ABB RobotStudio station: PickAndPlace_ManipulatorRobot.rspag

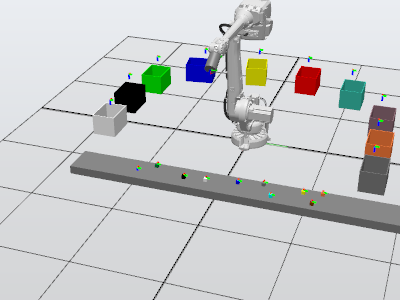
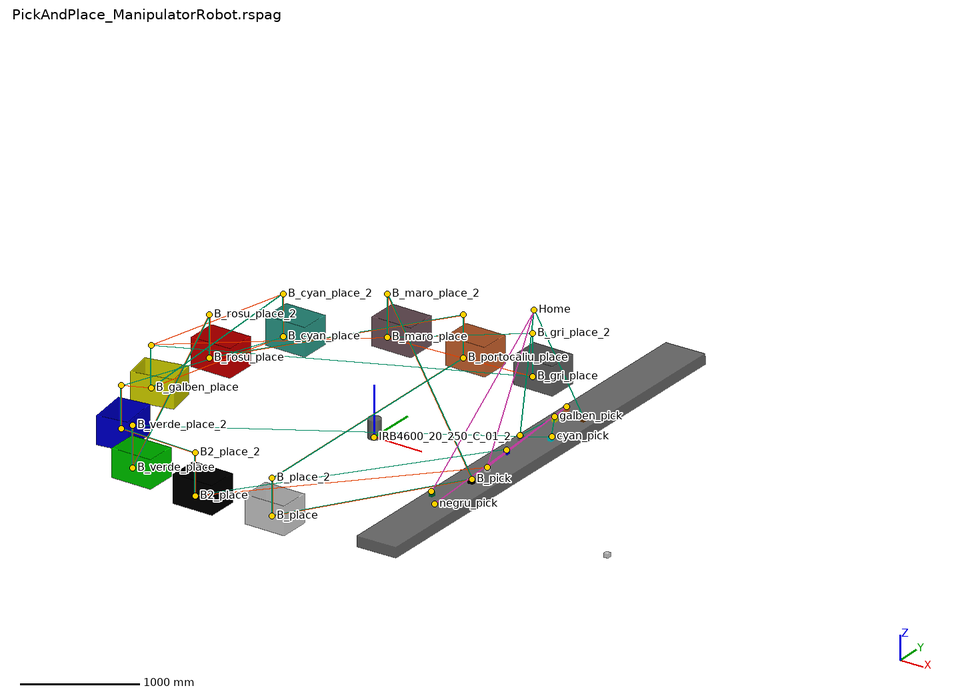
[picture v1: parts stored in the station drawn from their meshes, with robot base, taught points and paths (robot models come from the ABB library and are not in the file)]
--- station ---
Station Tema1 (saved by RobotStudio 24.3.10958.1)
Controller Controller1
  mechanical unit ROB_1: IRB4600_20_250_C_01_2, 6 joints, base frame (0, 0, 0) mm
Layout (positions relative to the parent item):
  - Container [part] at (-1892.47, -1896.95, 0) mm, size 400 x 300 x 270 mm
  - Container_2 [part] at (-161.95, 1479.58, 0) mm, size 400 x 300 x 270 mm
  - Container_4 [part] at (-1211.54, -114.6, 0) mm, rotated rx 0 ry 0 rz -168.57 deg, size 400 x 300 x 270 mm
  - Container_5 [part] at (-1951.65, -525.59, 0) mm, rotated rx 0 ry 0 rz -82.41 deg, size 400 x 300 x 270 mm
  - Cutia_alba [part] at (-473.04, -1981.87, 0) mm, size 400 x 300 x 270 mm
  - Container_7 [part] at (-1188.6, -2007.67, 0) mm, size 400 x 300 x 270 mm
  - Container_8 [part] at (-1549.29, 1401.48, 0) mm, size 400 x 300 x 270 mm
  - Container_9 [part] at (-2281.34, 903.83, 0) mm, size 400 x 300 x 270 mm
  - Container_10 [part] at (-2561.63, 214.84, 0) mm, size 400 x 300 x 270 mm
  - Banda Transport [part] at (1467.9, -1784.42, 101.57) mm, rotated rx -180 ry 0.95 rz -180 deg, size 400 x 4500 x 100 mm
  - Container_11 [part] at (-833.57, 1452.99, 0) mm, size 400 x 300 x 270 mm
  - griper [mechanism] at (1479.11, 0, 1722.5) mm, rotated rx -180 ry 60 rz -180 deg
      TCP griper at (0, 0, 175) mm
      links: Part_3
  - orn [part] at (2566.83, 0, 745.86) mm, size 40 x 40 x 40 mm
  - cutia_neagra-alb [part] at (1281.21, -423.55, 138.52) mm, rotated rx 180 ry 0 rz 180 deg, size 40 x 40 x 40 mm
  - alba [part] at (1269.69, -164.67, 139.56) mm, rotated rx 180 ry 0 rz 180 deg, size 40 x 40 x 40 mm
  - albastra [part] at (1207.67, 200.37, 140.96) mm, rotated rx 180 ry 0 rz 180 deg, size 40 x 40 x 40 mm
  - cyan [part] at (1364.48, 621.04, 140.84) mm, rotated rx 180 ry 0 rz 180 deg, size 40 x 40 x 40 mm
  - galben [part] at (1176.16, 945.56, 137.64) mm, rotated rx 180 ry 0 rz 180 deg, size 40 x 40 x 40 mm
  - rosu [part], size 40 x 40 x 40 mm
  - IRB4600_20_250_C_01_2 [mechanism, from %ABB.RobotStudio.Models.IRB4600%\IRB4600_20_250_C_G_01.rslib] at (0, 0, 0) mm; joint values [0, 0, 0, 0, 0.5236, 0] (rad or m)
  - ComponentInstance [part], size 120 x 119.8 x 175 mm
    - griper [frame] at (0, 0, 175) mm
  - Source [smart component, from Components\Source.rslib]
      properties: Source=cutia_neagra-alb; Copy=(none); Parent=(none); Position=[1.293592 -0.42159 0.14]; Orientation=[3.14159265358979 1.22460635382238E-16 -3.14159265358979]; Transient=false; PhysicsBehavior=-1
  - Queue [smart component, from Components\Queue.rslib]
      properties: Back=(none); Front=(none); Queue={ec790d8d-a707-48b2-aa37-b034cf45e0fb}; NumberOfObjects=1
  - albastru [part] at (1150.15, 487.08, 139.03) mm, rotated rx 180 ry 0 rz 180 deg, size 40 x 40 x 40 mm
  - portocaliu [part] at (1148.4, 1157.8, 139.66) mm, rotated rx 180 ry 0 rz 180 deg, size 40 x 40 x 40 mm
  - verde [part] at (1149.52, -806.44, 135.72) mm, rotated rx 180 ry 0 rz 180 deg, size 40 x 40 x 40 mm
  - maro [part] at (1371.34, 1079.42, 137.09) mm, rotated rx 180 ry 0 rz 180 deg, size 40 x 40 x 40 mm
  - galben [smart component, from Components\Queue.rslib]
      properties: Back=(none); Front=(none); Queue=; NumberOfObjects=0
  - Queue_5 [smart component, from Components\Queue.rslib]
      properties: Back=(none); Front=(none); Queue=; NumberOfObjects=0
  - Queue_6 [smart component, from Components\Queue.rslib]
      properties: Back=(none); Front=(none); Queue=; NumberOfObjects=0
  - Queue_7 [smart component, from Components\Queue.rslib]
      properties: Back=(none); Front=(none); Queue=; NumberOfObjects=0
  - Queue_8 [smart component, from Components\Queue.rslib]
      properties: Back=(none); Front=(none); Queue=; NumberOfObjects=0
  - Queue_9 [smart component, from Components\Queue.rslib]
      properties: Back=(none); Front=(none); Queue=; NumberOfObjects=0
  - Queue_10 [smart component, from Components\Queue.rslib]
      properties: Back=(none); Front=(none); Queue=; NumberOfObjects=0
  - Source_2 [smart component, from Components\Source.rslib]
      properties: Source=galben; Copy=(none); Parent=(none); Position=[1.177356 0.946132 0.14]; Orientation=[3.14159265358979 0 -3.14159265358979]; Transient=false; PhysicsBehavior=-1
  - Queue_11 [smart component, from Components\Queue.rslib]
      properties: Back=(none); Front=(none); Queue=; NumberOfObjects=0
  - Source_3 [smart component, from Components\Source.rslib]
      properties: Source=alba; Copy=(none); Parent=(none); Position=[1.26763 -0.163594 0.14]; Orientation=[3.14159265358979 0 -3.14159265358979]; Transient=false; PhysicsBehavior=-1
  - Source_4 [smart component, from Components\Source.rslib]
      properties: Source=albastra; Copy=(none); Parent=(none); Position=[1.209286 0.198923 0.14]; Orientation=[3.14159265358979 0 -3.14159265358979]; Transient=false; PhysicsBehavior=-1
  - Source_5 [smart component, from Components\Source.rslib]
      properties: Source=cyan; Copy=(none); Parent=(none); Position=[1.375124 0.620638 0.14]; Orientation=[3.14159265358979 0 -3.14159265358979]; Transient=false; PhysicsBehavior=-1
  - Source_6 [smart component, from Components\Source.rslib]
      properties: Source=rosu; Copy=(none); Parent=(none); Position=[1.26763 -0.163594 0.14]; Orientation=[3.14159265358979 0 -3.14159265358979]; Transient=false; PhysicsBehavior=-1
  - Source_7 [smart component, from Components\Source.rslib]
      properties: Source=albastru; Copy=(none); Parent=(none); Position=[1.145869 0.485999 0.14]; Orientation=[3.14159265358979 0 -3.14159265358979]; Transient=false; PhysicsBehavior=-1
  - Source_8 [smart component, from Components\Source.rslib]
      properties: Source=portocaliu; Copy=(none); Parent=(none); Position=[1.149217 1.156287 0.14]; Orientation=[3.14159265358979 0 -3.14159265358979]; Transient=false; PhysicsBehavior=-1
  - Source_9 [smart component, from Components\Source.rslib]
      properties: Source=verde; Copy=(none); Parent=(none); Position=[1.148873 -0.806327 0.14]; Orientation=[3.14159265358979 0 -3.14159265358979]; Transient=false; PhysicsBehavior=-1
  - Source_10 [smart component, from Components\Source.rslib]
      properties: Source=maro; Copy=(none); Parent=(none); Position=[1.372614 1.078627 0.14]; Orientation=[3.14159265358979 0 -3.14159265358979]; Transient=false; PhysicsBehavior=-1
  - Queue_12 [smart component, from Components\Queue.rslib]
      properties: Back=(none); Front=(none); Queue=; NumberOfObjects=0
  - cutia_neagra-alb_270 [part] at (1293.59, -421.59, 140) mm, rotated rx 180 ry 0 rz 180 deg, size 40 x 40 x 40 mm
  - cutia_neagra-alb_1129 [part] at (1293.59, -421.59, 140) mm, rotated rx 180 ry 0 rz 180 deg, size 40 x 40 x 40 mm
Attachment: griper is attached to IRB4600_20_250_C_01_2 / Link6
EventTableEntry 4264: Group=, Trigger=aa_gripper 4265, Actions=[EventTableActionAttach 4266], Comment=, ActivationMode=2, Cyclic=false
EventTableTriggerIO 4265: IOValue=[1], IRC5Controller=? -1, Operator=0, SignalSource=Controller1 6006
EventTableActionAttach 4266: AttachmentParent=griper 1033, AttachmentChild=? -1, MountObject=true, Offset=[X=1, Y=0, Z=0, W=0, X=0, Y=1, Z=0, W=0, X=0, Y=0, Z=1, W=0, X=0, Y=0, Z=0, W=1], FlangeIndext=0, FindNearest=true
EventTableEntry 4267: Group=, Trigger=aa_gripper 4268, Actions=[EventTableActionDetach 4269], Comment=, ActivationMode=2, Cyclic=false
EventTableTriggerIO 4268: IOValue=[0], IRC5Controller=? -1, Operator=0, SignalSource=Controller1 6006
EventTableActionDetach 4269: AttachmentParent=griper 1033, AttachmentChild=? -1
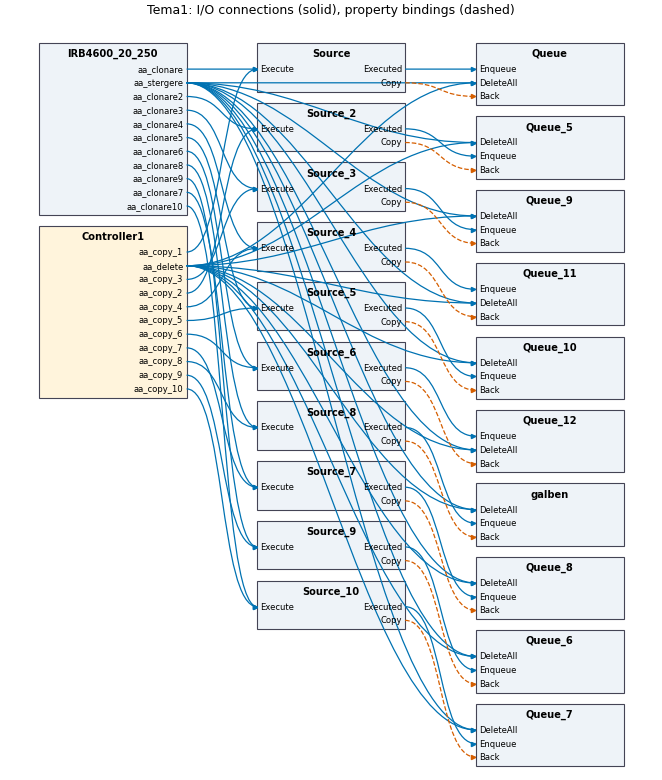
Station logic (signal -> signal, property => property):
  IRB4600_20_250.aa_clonare -> Source.Execute
  Source.Executed -> Queue.Enqueue
  IRB4600_20_250.aa_stergere -> Queue.DeleteAll
  IRB4600_20_250.aa_stergere -> Queue_5.DeleteAll
  Source_2.Executed -> Queue_5.Enqueue
  IRB4600_20_250.aa_stergere -> Queue_9.DeleteAll
  Source_3.Executed -> Queue_9.Enqueue
  Source_4.Executed -> Queue_11.Enqueue
  IRB4600_20_250.aa_stergere -> Queue_11.DeleteAll
  IRB4600_20_250.aa_stergere -> Queue_10.DeleteAll
  Source_5.Executed -> Queue_10.Enqueue
  Source_6.Executed -> Queue_12.Enqueue
  IRB4600_20_250.aa_stergere -> Queue_12.DeleteAll
  IRB4600_20_250.aa_stergere -> galben.DeleteAll
  IRB4600_20_250.aa_stergere -> Queue_6.DeleteAll
  IRB4600_20_250.aa_stergere -> Queue_7.DeleteAll
  IRB4600_20_250.aa_stergere -> Queue_8.DeleteAll
  Source_7.Executed -> Queue_8.Enqueue
  Source_8.Executed -> galben.Enqueue
  Source_9.Executed -> Queue_6.Enqueue
  Source_10.Executed -> Queue_7.Enqueue
  IRB4600_20_250.aa_clonare2 -> Source_2.Execute
  IRB4600_20_250.aa_clonare3 -> Source_3.Execute
  IRB4600_20_250.aa_clonare4 -> Source_4.Execute
  IRB4600_20_250.aa_clonare5 -> Source_5.Execute
  IRB4600_20_250.aa_clonare6 -> Source_6.Execute
  IRB4600_20_250.aa_clonare8 -> Source_8.Execute
  IRB4600_20_250.aa_clonare9 -> Source_9.Execute
  IRB4600_20_250.aa_clonare7 -> Source_7.Execute
  IRB4600_20_250.aa_clonare10 -> Source_10.Execute
  Controller1.aa_copy_1 -> Source.Execute
  Controller1.aa_delete -> Queue.DeleteAll
  Controller1.aa_delete -> Queue_5.DeleteAll
  Controller1.aa_delete -> Queue_9.DeleteAll
  Controller1.aa_delete -> Queue_11.DeleteAll
  Controller1.aa_delete -> galben.DeleteAll
  Controller1.aa_delete -> Queue_10.DeleteAll
  Controller1.aa_delete -> Queue_12.DeleteAll
  Controller1.aa_delete -> Queue_6.DeleteAll
  Controller1.aa_delete -> Queue_8.DeleteAll
  Controller1.aa_delete -> Queue_7.DeleteAll
  Controller1.aa_copy_3 -> Source_3.Execute
  Controller1.aa_copy_2 -> Source_2.Execute
  Controller1.aa_copy_4 -> Source_4.Execute
  Controller1.aa_copy_5 -> Source_5.Execute
  Controller1.aa_copy_6 -> Source_6.Execute
  Controller1.aa_copy_7 -> Source_7.Execute
  Controller1.aa_copy_8 -> Source_8.Execute
  Controller1.aa_copy_9 -> Source_9.Execute
  Controller1.aa_copy_10 -> Source_10.Execute
  Source.Copy => Queue.Back
  Source_2.Copy => Queue_5.Back
  Source_3.Copy => Queue_9.Back
  Source_4.Copy => Queue_11.Back
  Source_6.Copy => Queue_12.Back
  Source_5.Copy => Queue_10.Back
  Source_7.Copy => Queue_8.Back
  Source_8.Copy => galben.Back
  Source_9.Copy => Queue_6.Back
  Source_10.Copy => Queue_7.Back
Targets, tools, work objects and paths stored in the station and not in the controller backup, written as RAPID:
! task T_ROB1
MODULE Module1
  CONST robtarget Target_20:=[[1630.666635146,0.000000153,1634.999845105],[0.500000014,-0.000000026,0.866025396,-0.000000015],[0,-1,-1,0],[9E+09,9E+09,9E+09,9E+09,9E+09,9E+09]];
ENDMODULE


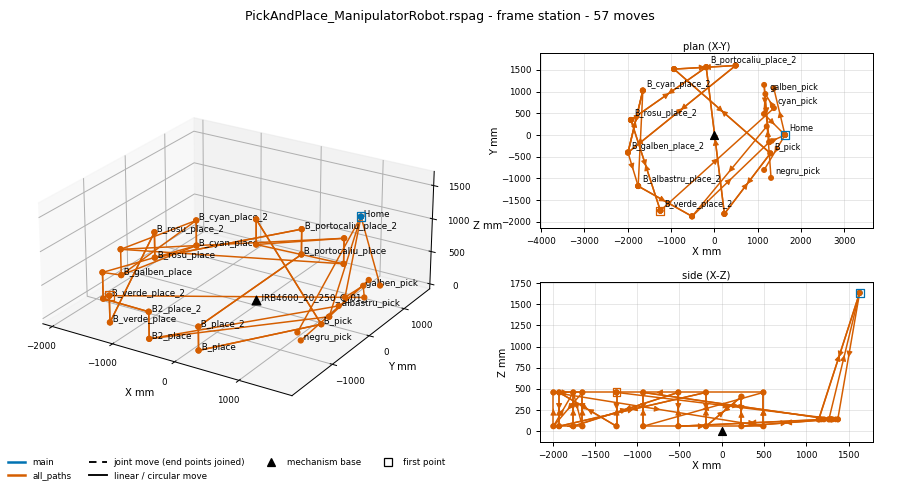
[picture p0: tool path of PickAndPlace_ManipulatorRobot.rspag in frame station, 57 of 71 moves have a stored position in this frame; points joined in program order, loops and branches not executed]
--- Backups/Controller1/RAPID/TASK1/PROGMOD/CalibData.mod ---
MODULE CalibData
    PERS tooldata griper:=[TRUE,[[0,0,175],[1,0,0,0]],[1,[0,0,1],[1,0,0,0],0,0,0]];
ENDMODULE

--- Backups/Controller1/RAPID/TASK1/PROGMOD/Module1.mod ---
MODULE Module1
    CONST robtarget Home:=[[1630.666611702,0.000000153,1634.999933868],[0.499999997,-0.000000012,0.866025406,-0.000000007],[0,-1,-1,0],[9E+09,9E+09,9E+09,9E+09,9E+09,9E+09]];
    CONST robtarget B_pick:=[[1293.592,-421.59,140],[0,0,1,0],[0,0,0,0],[9E+09,9E+09,9E+09,9E+09,9E+09,9E+09]];
    CONST robtarget B_place:=[[233.30176897,-1817.435857446,58.556],[0,0,1,0],[-1,0,-1,0],[9E+09,9E+09,9E+09,9E+09,9E+09,9E+09]];
    VAR robtarget my_pick;
    VAR robtarget my_place;
    VAR robtarget place;
    VAR robtarget clonare;
    VAR robtarget above_box;
    VAR num Array{2,3};
    CONST robtarget B2_pick:=[[1267.63,-163.594,140],[0,0,1,0],[-1,0,-1,0],[9E+09,9E+09,9E+09,9E+09,9E+09,9E+09]];
    CONST robtarget B2_place:=[[-512.842,-1875.439,58.556],[0,0,1,0],[-2,0,-2,0],[9E+09,9E+09,9E+09,9E+09,9E+09,9E+09]];
    CONST robtarget B_place_2:=[[233.30176897,-1817.435857446,408.556],[0,0,1,0],[-1,0,-1,0],[9E+09,9E+09,9E+09,9E+09,9E+09,9E+09]];
    CONST robtarget B_verde_place_2:=[[-1243.915,-1743.804,458.556],[0,0,1,0],[-2,0,-2,0],[9E+09,9E+09,9E+09,9E+09,9E+09,9E+09]];
    CONST robtarget B_verde_place:=[[-1243.915,-1743.804,58.556],[0,0,1,0],[-2,0,-2,0],[9E+09,9E+09,9E+09,9E+09,9E+09,9E+09]];
    CONST robtarget B_rosu_place_2:=[[-1923.035,348.607,458.556],[0,0,1,0],[1,0,1,0],[9E+09,9E+09,9E+09,9E+09,9E+09,9E+09]];
    CONST robtarget B_rosu_place:=[[-1923.035,348.607,58.556],[0,0,1,0],[1,0,1,0],[9E+09,9E+09,9E+09,9E+09,9E+09,9E+09]];
    CONST robtarget B_portocaliu_place_2:=[[-186.165,1564.222,458.556],[0,0,1,0],[0,0,0,0],[9E+09,9E+09,9E+09,9E+09,9E+09,9E+09]];
    CONST robtarget B_portocaliu_place:=[[-186.165,1564.222,58.556],[0,0,1,0],[0,0,0,0],[9E+09,9E+09,9E+09,9E+09,9E+09,9E+09]];
    CONST robtarget B_maro_place_2:=[[-928.266,1520.037,458.556],[0,0,1,0],[1,0,1,0],[9E+09,9E+09,9E+09,9E+09,9E+09,9E+09]];
    CONST robtarget B_maro_place:=[[-928.266,1520.037,58.556],[0,0,1,0],[1,0,1,0],[9E+09,9E+09,9E+09,9E+09,9E+09,9E+09]];
    CONST robtarget B_gri_place:=[[492.938,1602.646,58.556],[0,0,1,0],[0,0,0,0],[9E+09,9E+09,9E+09,9E+09,9E+09,9E+09]];
    CONST robtarget B_gri_place_2:=[[492.938,1602.646,458.556],[0,0,1,0],[0,0,0,0],[9E+09,9E+09,9E+09,9E+09,9E+09,9E+09]];
    CONST robtarget B_galben_place_2:=[[-1990.111,-403.463,458.556],[0,0,1,0],[-2,0,-2,0],[9E+09,9E+09,9E+09,9E+09,9E+09,9E+09]];
    CONST robtarget B_cyan_place_2:=[[-1647.649,1025.344,458.556],[0,0,1,0],[0,0,0,0],[9E+09,9E+09,9E+09,9E+09,9E+09,9E+09]];
    CONST robtarget B_cyan_place:=[[-1647.649,1025.344,58.556],[0,0,1,0],[0,0,0,0],[9E+09,9E+09,9E+09,9E+09,9E+09,9E+09]];
    CONST robtarget B_galben_place:=[[-1990.111,-403.463,58.556],[0,0,1,0],[-2,0,-2,0],[9E+09,9E+09,9E+09,9E+09,9E+09,9E+09]];
    CONST robtarget B_albastru_place_2:=[[-1755.688,-1177.677,458.556],[0,0,1,0],[-2,0,-2,0],[9E+09,9E+09,9E+09,9E+09,9E+09,9E+09]];
    CONST robtarget B_albastru_place:=[[-1755.688,-1177.677,58.556],[0,0,1,0],[-2,0,-2,0],[9E+09,9E+09,9E+09,9E+09,9E+09,9E+09]];
    CONST robtarget B2_place_2:=[[-512.842,-1875.439,458.556],[0,0,1,0],[-2,0,-2,0],[9E+09,9E+09,9E+09,9E+09,9E+09,9E+09]];
    CONST robtarget albastru_pick:=[[1209.286,198.923,140],[0,0,1,0],[0,0,0,0],[9E+09,9E+09,9E+09,9E+09,9E+09,9E+09]];
    CONST robtarget cyan_pick:=[[1375.124,620.638,140],[0,0,1,0],[0,0,0,0],[9E+09,9E+09,9E+09,9E+09,9E+09,9E+09]];
    CONST robtarget galben_pick:=[[1177.356,946.132,140],[0,0,1,0],[0,0,0,0],[9E+09,9E+09,9E+09,9E+09,9E+09,9E+09]];
    CONST robtarget gri_pick:=[[1145.869,485.999,140],[0,0,1,0],[0,0,0,0],[9E+09,9E+09,9E+09,9E+09,9E+09,9E+09]];
    CONST robtarget maro_pick:=[[1372.614,1078.627,140],[0,0,1,0],[0,0,0,0],[9E+09,9E+09,9E+09,9E+09,9E+09,9E+09]];
    CONST robtarget negru_pick:=[[1308.822,-989.177,140],[0,0,1,0],[-1,0,-1,0],[9E+09,9E+09,9E+09,9E+09,9E+09,9E+09]];
    CONST robtarget portocaliu_pick:=[[1149.217,1156.287,140],[0,0,1,0],[0,0,0,0],[9E+09,9E+09,9E+09,9E+09,9E+09,9E+09]];
    CONST robtarget Target_10:=[[1630.666635146,0.000000153,1634.999845105],[0.500000014,-0.000000026,0.866025396,-0.000000015],[0,-1,-1,0],[9E+09,9E+09,9E+09,9E+09,9E+09,9E+09]];
    CONST robtarget verde_pick:=[[1148.873,-806.327,140],[0,0,1,0],[-1,0,-1,0],[9E+09,9E+09,9E+09,9E+09,9E+09,9E+09]];
    CONST robtarget rosu_pick:=[[1267.63,-163.594,140],[0,0,1,0],[-1,0,-1,0],[9E+09,9E+09,9E+09,9E+09,9E+09,9E+09]];
!***********************************************************
    !
    ! Module:  Module1
    !
    ! Description:
    !   <Insert description here>
    !
    ! Author: Kiidal
    !
    ! Version: 1.0
    !
    !***********************************************************


    !***********************************************************
    !
    ! Procedure main
    !
    !   This is the entry point of your program
    !
    !***********************************************************
    PROC main()
    ! Add your code here

    MoveJ Home,v1000,z100,griper\WObj:=wobj0;

    WaitUntil(( Cutia_Alba = 1 ) OR ( cutia_Negro = 1 ) OR ( Cutia_Rosie = 1 ) OR ( Cutia_albastru = 1 ) OR
              ( Cutia_Verde = 1 ) OR ( Cutia_Galben = 1 ) OR ( Cutia_Cyan = 1 ) OR ( Cutia_Portocaliu = 1 ) OR
              ( Cutia_Gri = 1 ) OR ( Cutia_Maro = 1 ));

    IF Cutia_Alba = 1 THEN
        my_pick := B_pick;
        place := B_place;
        above_box := B_place_2;

          SetDO aa_copy_1,0;
    FOR i FROM 0 TO 7 DO

         SetDO aa_copy_1, 1;
         my_place := Offs(place, (i MOD 2) * 60, ((i DIV 2) MOD 2) * 60, (i DIV 4) * 40);

         New_Pick_and_place;


     SetDO aa_copy_1, 0;
    ENDFOR

    ELSEIF cutia_Negro = 1 THEN
        my_pick := B2_pick;
        place := B2_place;
        above_box := B2_place_2;

          SetDO aa_copy_3,0;
    FOR i FROM 0 TO 7 DO

         SetDO aa_copy_3, 1;
         my_place := Offs(place, (i MOD 2) * 60, ((i DIV 2) MOD 2) * 60, (i DIV 4) * 40);

         New_Pick_and_place;


     SetDO aa_copy_3, 0;

    ENDFOR

    ELSEIF Cutia_Rosie = 1 THEN
        my_pick := galben_pick;
        place := B_rosu_place;
        above_box := B_rosu_place_2;

          SetDO aa_copy_2,0;
    FOR i FROM 0 TO 7 DO

         SetDO aa_copy_2, 1;
         my_place := Offs(place, (i MOD 2) * 60, ((i DIV 2) MOD 2) * 60, (i DIV 4) * 40);

         New_Pick_and_place;


     SetDO aa_copy_2, 0;
    ENDFOR

    ELSEIF Cutia_albastru = 1 THEN
        my_pick := rosu_pick;
        place := B_albastru_place;
        above_box := B_albastru_place_2;

          SetDO aa_copy_6,0;
    FOR i FROM 0 TO 7 DO

         SetDO aa_copy_6, 1;
         my_place := Offs(place, (i MOD 2) * 60, ((i DIV 2) MOD 2) * 60, (i DIV 4) * 40);

         New_Pick_and_place;


     SetDO aa_copy_6, 0;
    ENDFOR

    ELSEIF Cutia_Verde = 1 THEN
        my_pick := albastru_pick;
        place := B_verde_place;
        above_box := B_verde_place_2;
          SetDO aa_copy_4,0;
    FOR i FROM 0 TO 7 DO

         SetDO aa_copy_4, 1;
         my_place := Offs(place, (i MOD 2) * 60, ((i DIV 2) MOD 2) * 60, (i DIV 4) * 40);

         New_Pick_and_place;


     SetDO aa_copy_4, 0;
    ENDFOR

    ELSEIF Cutia_Galben = 1 THEN
        my_pick := cyan_pick;
        place := B_galben_place;
        above_box := B_galben_place_2;
          SetDO aa_copy_5,0;
    FOR i FROM 0 TO 7 DO

         SetDO aa_copy_5, 1;
         my_place := Offs(place, (i MOD 2) * 60, ((i DIV 2) MOD 2) * 60, (i DIV 4) * 40);

         New_Pick_and_place;


     SetDO aa_copy_5, 0;
    ENDFOR

    ELSEIF Cutia_Cyan = 1 THEN
        my_pick := gri_pick;
        place := B_cyan_place;
        above_box := B_cyan_place_2;
          SetDO aa_copy_7,0;
    FOR i FROM 0 TO 7 DO

         SetDO aa_copy_7, 1;
         my_place := Offs(place, (i MOD 2) * 60, ((i DIV 2) MOD 2) * 60, (i DIV 4) * 40);

         New_Pick_and_place;


     SetDO aa_copy_7, 0;
    ENDFOR

    ELSEIF Cutia_Portocaliu = 1 THEN
        my_pick := maro_pick;
        place := B_portocaliu_place;
        above_box := B_portocaliu_place_2;
          SetDO aa_copy_10,0;
    FOR i FROM 0 TO 7 DO

         SetDO aa_copy_10, 1;
         my_place := Offs(place, (i MOD 2) * 60, ((i DIV 2) MOD 2) * 60, (i DIV 4) * 40);

         New_Pick_and_place;


     SetDO aa_copy_10, 0;
    ENDFOR

    ELSEIF Cutia_Gri = 1 THEN
        my_pick := portocaliu_pick;
        place := B_gri_place;
        above_box := B_gri_place_2;
          SetDO aa_copy_8,0;
    FOR i FROM 0 TO 7 DO

         SetDO aa_copy_8, 1;
         my_place := Offs(place, (i MOD 2) * 60, ((i DIV 2) MOD 2) * 60, (i DIV 4) * 40);

         New_Pick_and_place;


     SetDO aa_copy_8, 0;
    ENDFOR

    ELSEIF Cutia_Maro =1 THEN
        my_pick := verde_pick;
        place := B_maro_place;
        above_box := B_maro_place_2;
          SetDO aa_copy_9,0;
    FOR i FROM 0 TO 7 DO

         SetDO aa_copy_9, 1;
         my_place := Offs(place, (i MOD 2) * 60, ((i DIV 2) MOD 2) * 60, (i DIV 4) * 40);

         New_Pick_and_place;

     SetDO aa_copy_9, 0;
    ENDFOR

    ENDIF


    SetDO aa_delete, 0;

    MoveJ Home,v1000,z100,griper\WObj:=wobj0;

    SetDO aa_delete, 1;

    ENDPROC


    PROC New_Pick_and_place()

        SetDo aa_gripper,0;

        MoveJ offs(my_pick,0,0,100),v1000,fine,griper\WObj:=wobj0;
        MoveL my_pick,v1000,fine,griper\WObj:=wobj0;
        SetDO aa_gripper,1;
        WaitTime 0.5;
        MoveL offs(my_pick,0,0,100),v1000,fine,griper\WObj:=wobj0;

        MoveJ offs(above_box,0,0,100),v1000,fine,griper\WObj:=wobj0;
        MoveL above_box,v1000,fine,griper\WObj:=wobj0;

        MoveJ offs(my_place,0,0,100),v1000,fine,griper\WObj:=wobj0;
        MoveL my_place,v1000,fine,griper\WObj:=wobj0;
        SetDo aa_gripper,0;
        MoveL offs(my_place,0,0,100),v1000,fine,griper\WObj:=wobj0;

        WaitTime 0.5;
        MoveL offs(above_box,0,0,100),v1000,fine,griper\WObj:=wobj0;
        MoveL above_box,v1000,fine,griper\WObj:=wobj0;

    ENDPROC
    PROC all_paths()
        MoveL B_verde_place_2,v1000,z100,griper\WObj:=wobj0;
        MoveL B_verde_place_2,v1000,z100,griper\WObj:=wobj0;
        MoveL B_verde_place,v1000,z100,griper\WObj:=wobj0;
        MoveL B_rosu_place_2,v1000,z100,griper\WObj:=wobj0;
        MoveL B_rosu_place,v1000,z100,griper\WObj:=wobj0;
        MoveL B_portocaliu_place_2,v1000,z100,griper\WObj:=wobj0;
        MoveL B_portocaliu_place,v1000,z100,griper\WObj:=wobj0;
        MoveL B_place_2,v1000,z100,griper\WObj:=wobj0;
        MoveL B_place,v1000,z100,griper\WObj:=wobj0;
        MoveL B_pick,v1000,z100,griper\WObj:=wobj0;
        MoveL B_maro_place_2,v1000,z100,griper\WObj:=wobj0;
        MoveL B_maro_place,v1000,z100,griper\WObj:=wobj0;
        MoveL B_gri_place,v1000,z100,griper\WObj:=wobj0;
        MoveL B_gri_place_2,v1000,z100,griper\WObj:=wobj0;
        MoveL B_galben_place_2,v1000,z100,griper\WObj:=wobj0;
        MoveL B_cyan_place_2,v1000,z100,griper\WObj:=wobj0;
        MoveL B_cyan_place,v1000,z100,griper\WObj:=wobj0;
        MoveL B_galben_place,v1000,z100,griper\WObj:=wobj0;
        MoveL B_albastru_place_2,v1000,z100,griper\WObj:=wobj0;
        MoveL B_albastru_place,v1000,z100,griper\WObj:=wobj0;
        MoveL B2_place_2,v1000,z100,griper\WObj:=wobj0;
        MoveL B2_place,v1000,z100,griper\WObj:=wobj0;
        MoveL rosu_pick,v1000,z100,griper\WObj:=wobj0;
        MoveL above_box,v1000,z100,griper\WObj:=wobj0;
        MoveL above_box,v1000,z100,griper\WObj:=wobj0;
        MoveL albastru_pick,v1000,z100,griper\WObj:=wobj0;
        MoveL B2_place,v1000,z100,griper\WObj:=wobj0;
        MoveL B2_place_2,v1000,z100,griper\WObj:=wobj0;
        MoveL B_albastru_place,v1000,z100,griper\WObj:=wobj0;
        MoveL B_albastru_place_2,v1000,z100,griper\WObj:=wobj0;
        MoveL B_cyan_place,v1000,z100,griper\WObj:=wobj0;
        MoveL B_cyan_place_2,v1000,z100,griper\WObj:=wobj0;
        MoveL B_galben_place,v1000,z100,griper\WObj:=wobj0;
        MoveL B_galben_place_2,v1000,z100,griper\WObj:=wobj0;
        MoveL B_gri_place,v1000,z100,griper\WObj:=wobj0;
        MoveL B_gri_place_2,v1000,z100,griper\WObj:=wobj0;
        MoveL B_maro_place,v1000,z100,griper\WObj:=wobj0;
        MoveL B_maro_place_2,v1000,z100,griper\WObj:=wobj0;
        MoveL B_pick,v1000,z100,griper\WObj:=wobj0;
        MoveL B_place,v1000,z100,griper\WObj:=wobj0;
        MoveL B_place_2,v1000,z100,griper\WObj:=wobj0;
        MoveL B_portocaliu_place,v1000,z100,griper\WObj:=wobj0;
        MoveL B_portocaliu_place_2,v1000,z100,griper\WObj:=wobj0;
        MoveL B_rosu_place,v1000,z100,griper\WObj:=wobj0;
        MoveL B_rosu_place_2,v1000,z100,griper\WObj:=wobj0;
        MoveL B_verde_place,v1000,z100,griper\WObj:=wobj0;
        MoveL B_verde_place_2,v1000,z100,griper\WObj:=wobj0;
        MoveL cyan_pick,v1000,z100,griper\WObj:=wobj0;
        MoveL galben_pick,v1000,z100,griper\WObj:=wobj0;
        MoveL gri_pick,v1000,z100,griper\WObj:=wobj0;
        MoveL Home,v1000,z100,griper\WObj:=wobj0;
        MoveL maro_pick,v1000,z100,griper\WObj:=wobj0;
        MoveL my_pick,v1000,z100,griper\WObj:=wobj0;
        MoveL my_place,v1000,z100,griper\WObj:=wobj0;
        MoveL negru_pick,v1000,z100,griper\WObj:=wobj0;
        MoveL portocaliu_pick,v1000,z100,griper\WObj:=wobj0;
        MoveL rosu_pick,v1000,z100,griper\WObj:=wobj0;
        MoveL Target_10,v1000,z100,griper\WObj:=wobj0;
        MoveL verde_pick,v1000,z100,griper\WObj:=wobj0;
    ENDPROC



ENDMODULE

--- Backups/Controller1/SYSPAR/EIO.cfg ---
EIO:CFG_1.0:6:1::
#
EIO_SIGNAL:

      -Name "aa_gripper" -SignalType "DO" -Access "All"

      -Name "aa_copy_1" -SignalType "DO"

      -Name "aa_copy_2" -SignalType "DO"

      -Name "aa_copy_3" -SignalType "DO"

      -Name "aa_copy_4" -SignalType "DO"

      -Name "aa_copy_5" -SignalType "DO"

      -Name "aa_copy_6" -SignalType "DO"

      -Name "aa_copy_7" -SignalType "DO"

      -Name "aa_copy_8" -SignalType "DO"

      -Name "aa_copy_9" -SignalType "DO"

      -Name "aa_copy_10" -SignalType "DO"

      -Name "aa_delete" -SignalType "DO"

      -Name "Cutia_Alba" -SignalType "DI"

      -Name "Cutia_albastru" -SignalType "DI"

      -Name "Cutia_Cyan" -SignalType "DI"

      -Name "Cutia_Gri" -SignalType "DI"

      -Name "Cutia_Maro" -SignalType "DI"

      -Name "Cutia_Portocaliu" -SignalType "DI"

      -Name "Cutia_Rosie" -SignalType "DI"

      -Name "Cutia_Verde" -SignalType "DI"

      -Name "cutia_Negro" -SignalType "DI"

      -Name "Cutia_Galben" -SignalType "DI"
